Fanuc KAREL source: kt00444.KL

-- PROVISIONAL review KL for V770-1; original PC SHA256 1df7988e9a34a75460a0f83f6fce9d7c52ece00f6a60adf0854f708dfb2c483d
-- Incomplete behavior may be omitted. Consult companion uncertainty JSON. Do not deploy.
PROGRAM KT00444
%NOLOCKGROUP
VAR
  R1 : REAL
  OUT : BOOLEAN
-- UNRESOLVED_DECL H2 type=002017
BEGIN
  -- UNRESOLVED_PC offsets 5-16; opcodes 2E,23
  -- UNRESOLVED_PC offsets 21-35; opcodes 2E,22,9D,33,B4
  -- UNRESOLVED_PC offsets 40-63; opcodes 21,22,9D,33,B3,64,72,23
  -- UNRESOLVED_PC offsets 68-72; opcodes 7F
END KT00444
